DATA_BLOCK "IEC_Counter_0_DB"
{InstructionName := 'IEC_COUNTER';
 LibVersion := '1.0';
 S7_Optimized_Access := 'TRUE' }
AUTHOR : Simatic
FAMILY : IEC
NAME : CNTR
VERSION : 1.0
IEC_COUNTER

BEGIN

END_DATA_BLOCK

